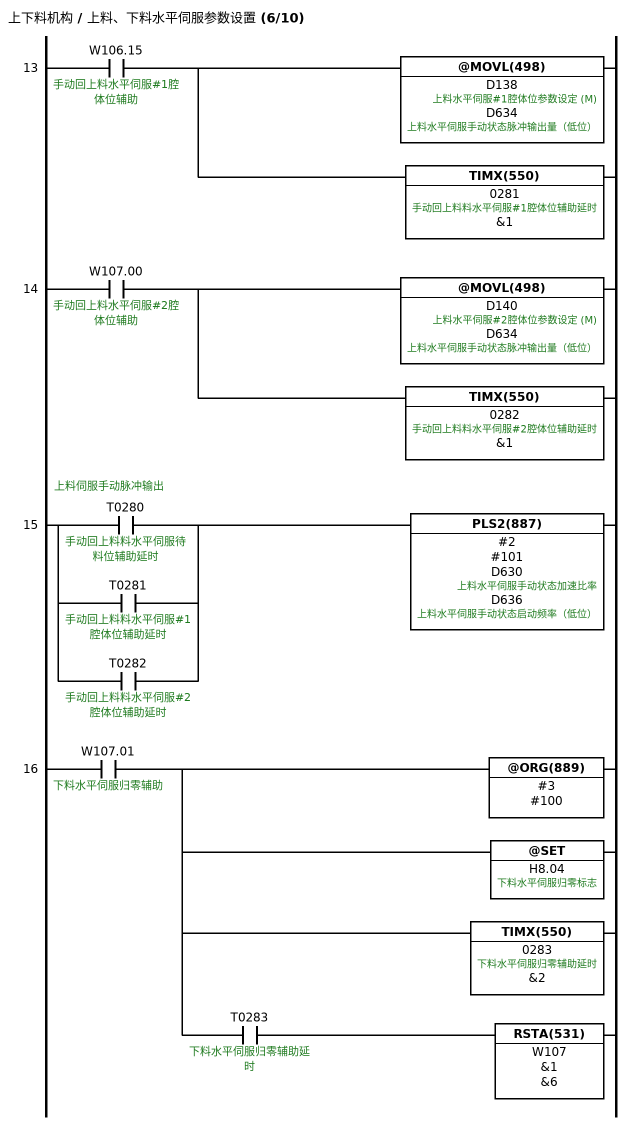
; [picture p216: 上下料机构 / 上料、下料水平伺服参数设置, rungs 13-16]
; rung 13
LD W106.15  ; 手动回上料水平伺服#1腔体位辅助
@MOVL(498) D138 D634  ; 上料水平伺服#1腔体位参数设定 (M), 上料水平伺服手动状态脉冲输出量（低位）
TIMX(550) 0281 &1  ; 手动回上料料水平伺服#1腔体位辅助延时
; rung 14
LD W107.00  ; 手动回上料水平伺服#2腔体位辅助
@MOVL(498) D140 D634  ; 上料水平伺服#2腔体位参数设定 (M), 上料水平伺服手动状态脉冲输出量（低位）
TIMX(550) 0282 &1  ; 手动回上料料水平伺服#2腔体位辅助延时
; rung 15: 上料伺服手动脉冲输出
LD T0280  ; 手动回上料料水平伺服待料位辅助延时
OR T0281  ; 手动回上料料水平伺服#1腔体位辅助延时
OR T0282  ; 手动回上料料水平伺服#2腔体位辅助延时
PLS2(887) #2 #101 D630 D636  ; 上料水平伺服手动状态加速比率, 上料水平伺服手动状态启动频率（低位）
; rung 16
LD W107.01  ; 下料水平伺服归零辅助
@ORG(889) #3 #100
@SET H8.04  ; 下料水平伺服归零标志
TIMX(550) 0283 &2  ; 下料水平伺服归零辅助延时
AND T0283  ; 下料水平伺服归零辅助延时
RSTA(531) W107 &1 &6

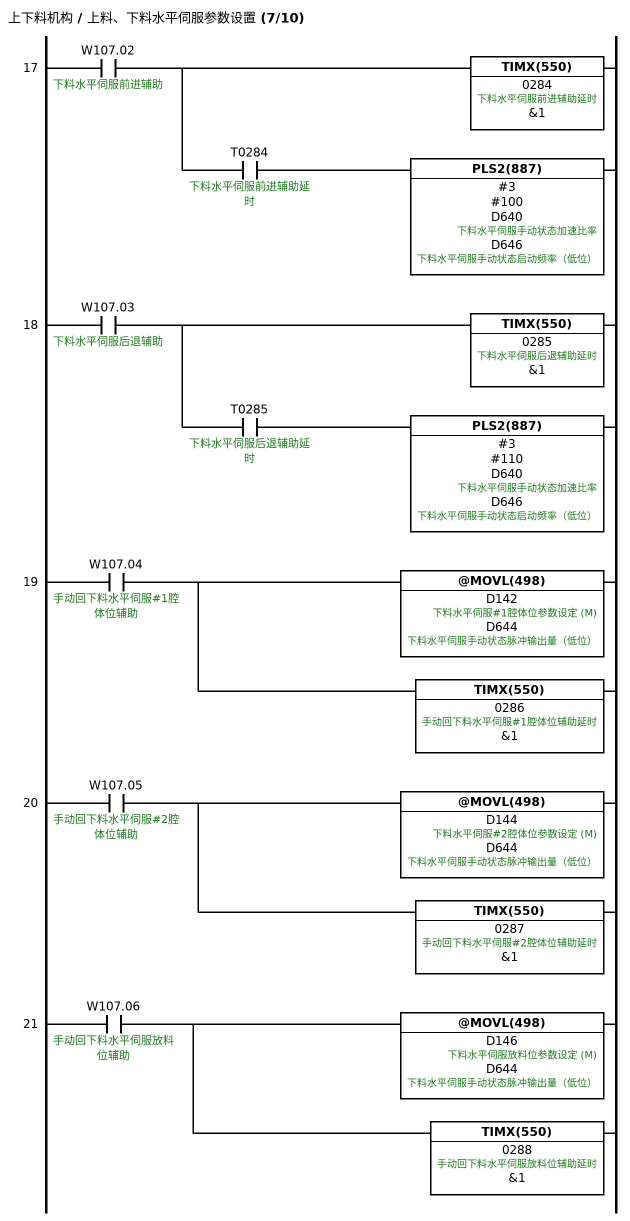
; rung 17
LD W107.02  ; 下料水平伺服前进辅助
TIMX(550) 0284 &1  ; 下料水平伺服前进辅助延时
AND T0284  ; 下料水平伺服前进辅助延时
PLS2(887) #3 #100 D640 D646  ; 下料水平伺服手动状态加速比率, 下料水平伺服手动状态启动频率（低位）
; rung 18
LD W107.03  ; 下料水平伺服后退辅助
TIMX(550) 0285 &1  ; 下料水平伺服后退辅助延时
AND T0285  ; 下料水平伺服后退辅助延时
PLS2(887) #3 #110 D640 D646  ; 下料水平伺服手动状态加速比率, 下料水平伺服手动状态启动频率（低位）
; rung 19
LD W107.04  ; 手动回下料水平伺服#1腔体位辅助
@MOVL(498) D142 D644  ; 下料水平伺服#1腔体位参数设定 (M), 下料水平伺服手动状态脉冲输出量（低位）
TIMX(550) 0286 &1  ; 手动回下料水平伺服#1腔体位辅助延时
; rung 20
LD W107.05  ; 手动回下料水平伺服#2腔体位辅助
@MOVL(498) D144 D644  ; 下料水平伺服#2腔体位参数设定 (M), 下料水平伺服手动状态脉冲输出量（低位）
TIMX(550) 0287 &1  ; 手动回下料水平伺服#2腔体位辅助延时
; rung 21
LD W107.06  ; 手动回下料水平伺服放料位辅助
@MOVL(498) D146 D644  ; 下料水平伺服放料位参数设定 (M), 下料水平伺服手动状态脉冲输出量（低位）
TIMX(550) 0288 &1  ; 手动回下料水平伺服放料位辅助延时

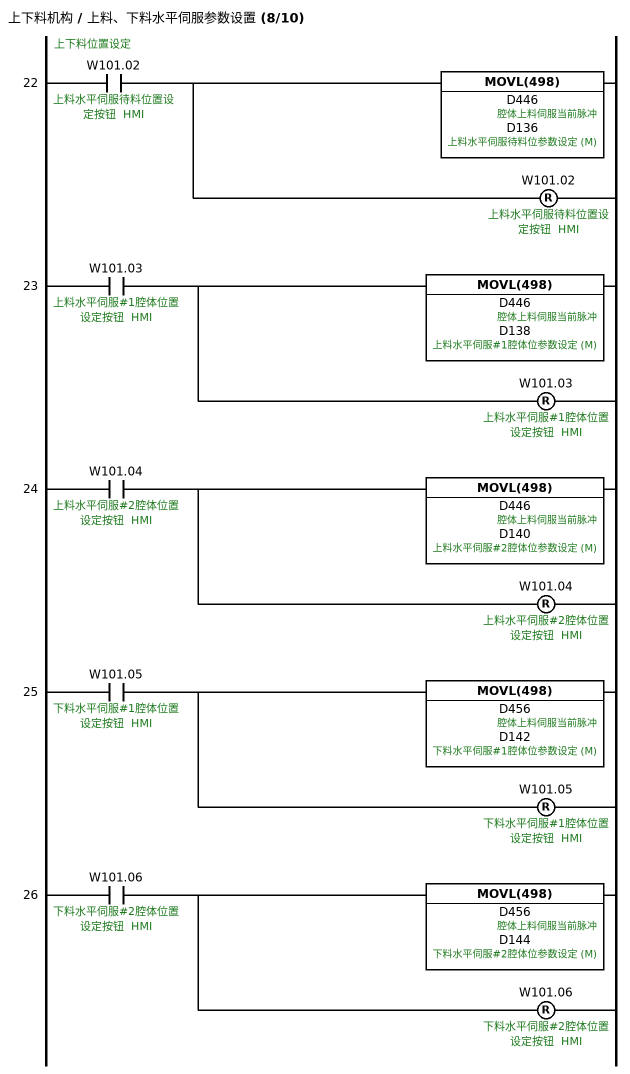
; rung 22: 上下料位置设定
LD W101.02  ; 上料水平伺服待料位置设定按钮  HMI
MOVL(498) D446 D136  ; 腔体上料伺服当前脉冲, 上料水平伺服待料位参数设定 (M)
RSET W101.02  ; 上料水平伺服待料位置设定按钮  HMI
; rung 23
LD W101.03  ; 上料水平伺服#1腔体位置设定按钮  HMI
MOVL(498) D446 D138  ; 腔体上料伺服当前脉冲, 上料水平伺服#1腔体位参数设定 (M)
RSET W101.03  ; 上料水平伺服#1腔体位置设定按钮  HMI
; rung 24
LD W101.04  ; 上料水平伺服#2腔体位置设定按钮  HMI
MOVL(498) D446 D140  ; 腔体上料伺服当前脉冲, 上料水平伺服#2腔体位参数设定 (M)
RSET W101.04  ; 上料水平伺服#2腔体位置设定按钮  HMI
; rung 25
LD W101.05  ; 下料水平伺服#1腔体位置设定按钮  HMI
MOVL(498) D456 D142  ; 腔体上料伺服当前脉冲, 下料水平伺服#1腔体位参数设定 (M)
RSET W101.05  ; 下料水平伺服#1腔体位置设定按钮  HMI
; rung 26
LD W101.06  ; 下料水平伺服#2腔体位置设定按钮  HMI
MOVL(498) D456 D144  ; 腔体上料伺服当前脉冲, 下料水平伺服#2腔体位参数设定 (M)
RSET W101.06  ; 下料水平伺服#2腔体位置设定按钮  HMI

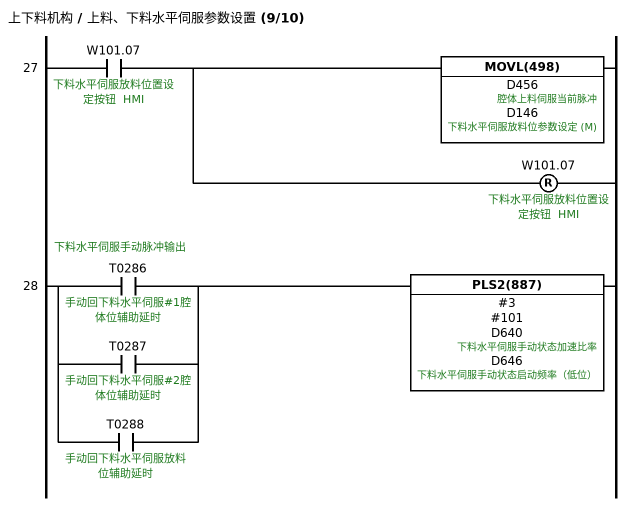
; rung 27
LD W101.07  ; 下料水平伺服放料位置设定按钮  HMI
MOVL(498) D456 D146  ; 腔体上料伺服当前脉冲, 下料水平伺服放料位参数设定 (M)
RSET W101.07  ; 下料水平伺服放料位置设定按钮  HMI
; rung 28: 下料水平伺服手动脉冲输出
LD T0286  ; 手动回下料水平伺服#1腔体位辅助延时
OR T0287  ; 手动回下料水平伺服#2腔体位辅助延时
OR T0288  ; 手动回下料水平伺服放料位辅助延时
PLS2(887) #3 #101 D640 D646  ; 下料水平伺服手动状态加速比率, 下料水平伺服手动状态启动频率（低位）

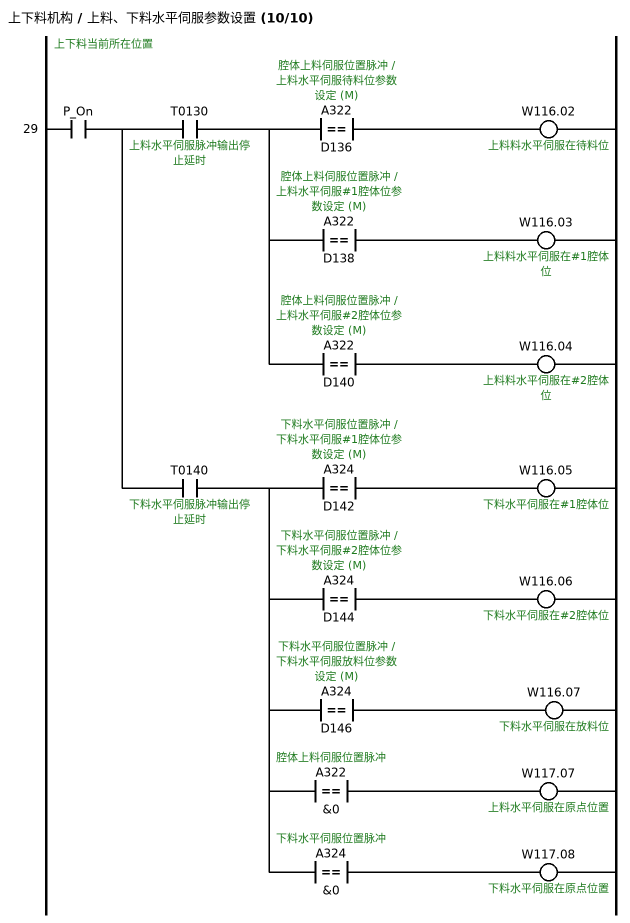
; rung 29: 上下料当前所在位置
LD P_On
OUT TR0
AND T0130  ; 上料水平伺服脉冲输出停止延时
OUT TR1
AND=SL(303) A322 D136  ; 腔体上料伺服位置脉冲, 上料水平伺服待料位参数设定 (M)
OUT W116.02  ; 上料料水平伺服在待料位
LD TR1
AND=SL(303) A322 D138  ; 腔体上料伺服位置脉冲, 上料水平伺服#1腔体位参数设定 (M)
OUT W116.03  ; 上料料水平伺服在#1腔体位
LD TR1
AND=SL(303) A322 D140  ; 腔体上料伺服位置脉冲, 上料水平伺服#2腔体位参数设定 (M)
OUT W116.04  ; 上料料水平伺服在#2腔体位
LD TR0
AND T0140  ; 下料水平伺服脉冲输出停止延时
OUT TR0
AND=SL(303) A324 D142  ; 下料水平伺服位置脉冲, 下料水平伺服#1腔体位参数设定 (M)
OUT W116.05  ; 下料水平伺服在#1腔体位
LD TR0
AND=SL(303) A324 D144  ; 下料水平伺服位置脉冲, 下料水平伺服#2腔体位参数设定 (M)
OUT W116.06  ; 下料水平伺服在#2腔体位
LD TR0
AND=SL(303) A324 D146  ; 下料水平伺服位置脉冲, 下料水平伺服放料位参数设定 (M)
OUT W116.07  ; 下料水平伺服在放料位
LD TR0
AND=SL(303) A322 &0  ; 腔体上料伺服位置脉冲
OUT W117.07  ; 上料水平伺服在原点位置
LD TR0
AND=SL(303) A324 &0  ; 下料水平伺服位置脉冲
OUT W117.08  ; 下料水平伺服在原点位置

### Section 工站复位

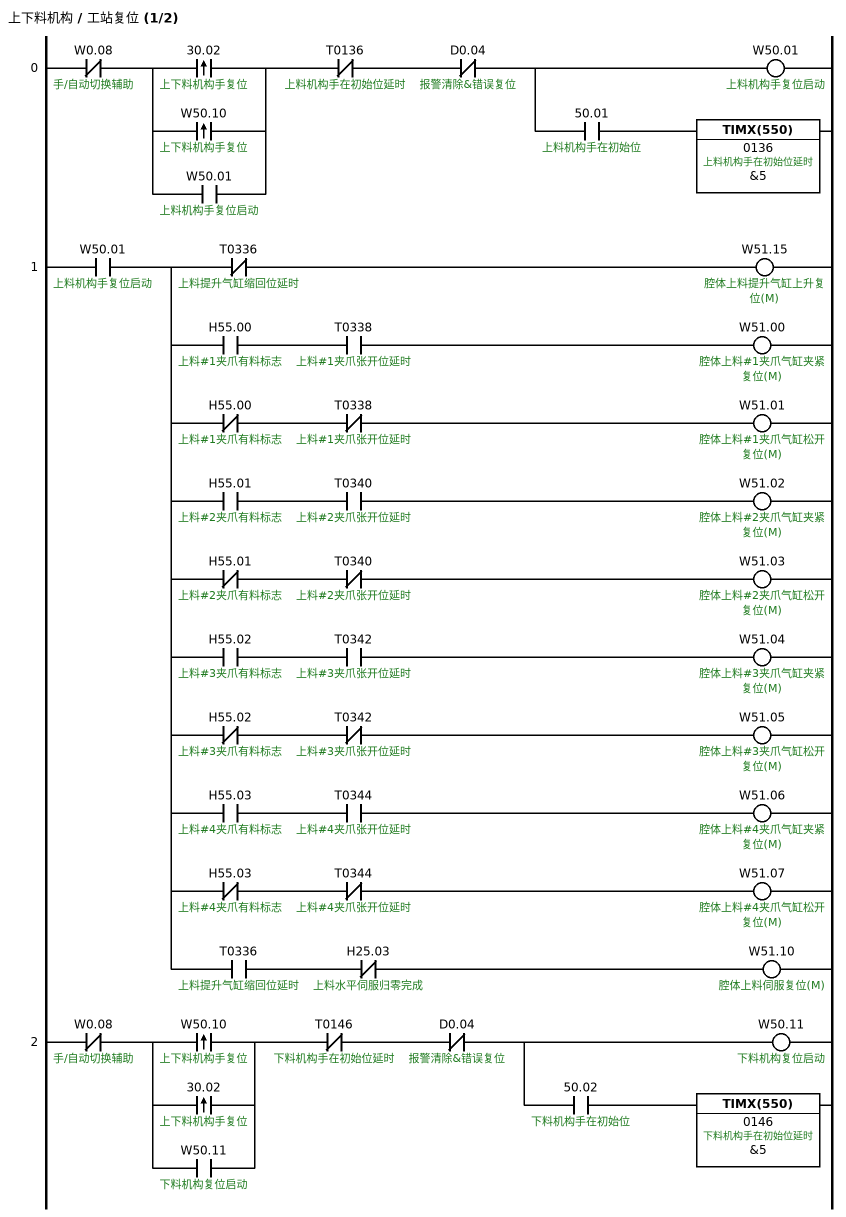
; rung 0
LDNOT W0.08  ; 手/自动切换辅助
@LD 30.02  ; 上下料机构手复位
@OR W50.10  ; 上下料机构手复位
OR W50.01  ; 上料机构手复位启动
ANDLD
ANDNOT T0136  ; 上料机构手在初始位延时
ANDNOT D0.04  ; 报警清除&错误复位
OUT W50.01  ; 上料机构手复位启动
AND 50.01  ; 上料机构手在初始位
TIMX(550) 0136 &5  ; 上料机构手在初始位延时
; rung 1
LD W50.01  ; 上料机构手复位启动
OUT TR0
ANDNOT T0336  ; 上料提升气缸缩回位延时
OUT W51.15  ; 腔体上料提升气缸上升复位(M)
LD TR0
AND H55.00  ; 上料#1夹爪有料标志
AND T0338  ; 上料#1夹爪张开位延时
OUT W51.00  ; 腔体上料#1夹爪气缸夹紧复位(M)
LD TR0
ANDNOT H55.00  ; 上料#1夹爪有料标志
ANDNOT T0338  ; 上料#1夹爪张开位延时
OUT W51.01  ; 腔体上料#1夹爪气缸松开复位(M)
LD TR0
AND H55.01  ; 上料#2夹爪有料标志
AND T0340  ; 上料#2夹爪张开位延时
OUT W51.02  ; 腔体上料#2夹爪气缸夹紧复位(M)
LD TR0
ANDNOT H55.01  ; 上料#2夹爪有料标志
ANDNOT T0340  ; 上料#2夹爪张开位延时
OUT W51.03  ; 腔体上料#2夹爪气缸松开复位(M)
LD TR0
AND H55.02  ; 上料#3夹爪有料标志
AND T0342  ; 上料#3夹爪张开位延时
OUT W51.04  ; 腔体上料#3夹爪气缸夹紧复位(M)
LD TR0
ANDNOT H55.02  ; 上料#3夹爪有料标志
ANDNOT T0342  ; 上料#3夹爪张开位延时
OUT W51.05  ; 腔体上料#3夹爪气缸松开复位(M)
LD TR0
AND H55.03  ; 上料#4夹爪有料标志
AND T0344  ; 上料#4夹爪张开位延时
OUT W51.06  ; 腔体上料#4夹爪气缸夹紧复位(M)
LD TR0
ANDNOT H55.03  ; 上料#4夹爪有料标志
ANDNOT T0344  ; 上料#4夹爪张开位延时
OUT W51.07  ; 腔体上料#4夹爪气缸松开复位(M)
LD TR0
AND T0336  ; 上料提升气缸缩回位延时
ANDNOT H25.03  ; 上料水平伺服归零完成
OUT W51.10  ; 腔体上料伺服复位(M)
; rung 2
LDNOT W0.08  ; 手/自动切换辅助
@LD W50.10  ; 上下料机构手复位
@OR 30.02  ; 上下料机构手复位
OR W50.11  ; 下料机构复位启动
ANDLD
ANDNOT T0146  ; 下料机构手在初始位延时
ANDNOT D0.04  ; 报警清除&错误复位
OUT W50.11  ; 下料机构复位启动
AND 50.02  ; 下料机构手在初始位
TIMX(550) 0146 &5  ; 下料机构手在初始位延时

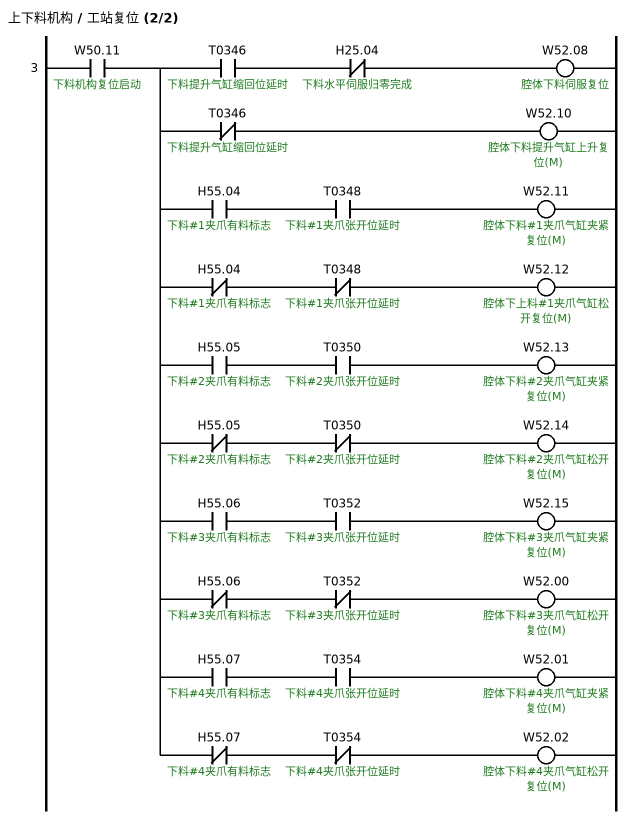
; rung 3
LD W50.11  ; 下料机构复位启动
OUT TR0
AND T0346  ; 下料提升气缸缩回位延时
ANDNOT H25.04  ; 下料水平伺服归零完成
OUT W52.08  ; 腔体下料伺服复位
LD TR0
ANDNOT T0346  ; 下料提升气缸缩回位延时
OUT W52.10  ; 腔体下料提升气缸上升复位(M)
LD TR0
AND H55.04  ; 下料#1夹爪有料标志
AND T0348  ; 下料#1夹爪张开位延时
OUT W52.11  ; 腔体下料#1夹爪气缸夹紧复位(M)
LD TR0
ANDNOT H55.04  ; 下料#1夹爪有料标志
ANDNOT T0348  ; 下料#1夹爪张开位延时
OUT W52.12  ; 腔体下上料#1夹爪气缸松开复位(M)
LD TR0
AND H55.05  ; 下料#2夹爪有料标志
AND T0350  ; 下料#2夹爪张开位延时
OUT W52.13  ; 腔体下料#2夹爪气缸夹紧复位(M)
LD TR0
ANDNOT H55.05  ; 下料#2夹爪有料标志
ANDNOT T0350  ; 下料#2夹爪张开位延时
OUT W52.14  ; 腔体下料#2夹爪气缸松开复位(M)
LD TR0
AND H55.06  ; 下料#3夹爪有料标志
AND T0352  ; 下料#3夹爪张开位延时
OUT W52.15  ; 腔体下料#3夹爪气缸夹紧复位(M)
LD TR0
ANDNOT H55.06  ; 下料#3夹爪有料标志
ANDNOT T0352  ; 下料#3夹爪张开位延时
OUT W52.00  ; 腔体下料#3夹爪气缸松开复位(M)
LD TR0
AND H55.07  ; 下料#4夹爪有料标志
AND T0354  ; 下料#4夹爪张开位延时
OUT W52.01  ; 腔体下料#4夹爪气缸夹紧复位(M)
LD TR0
ANDNOT H55.07  ; 下料#4夹爪有料标志
ANDNOT T0354  ; 下料#4夹爪张开位延时
OUT W52.02  ; 腔体下料#4夹爪气缸松开复位(M)

### Section 指示灯

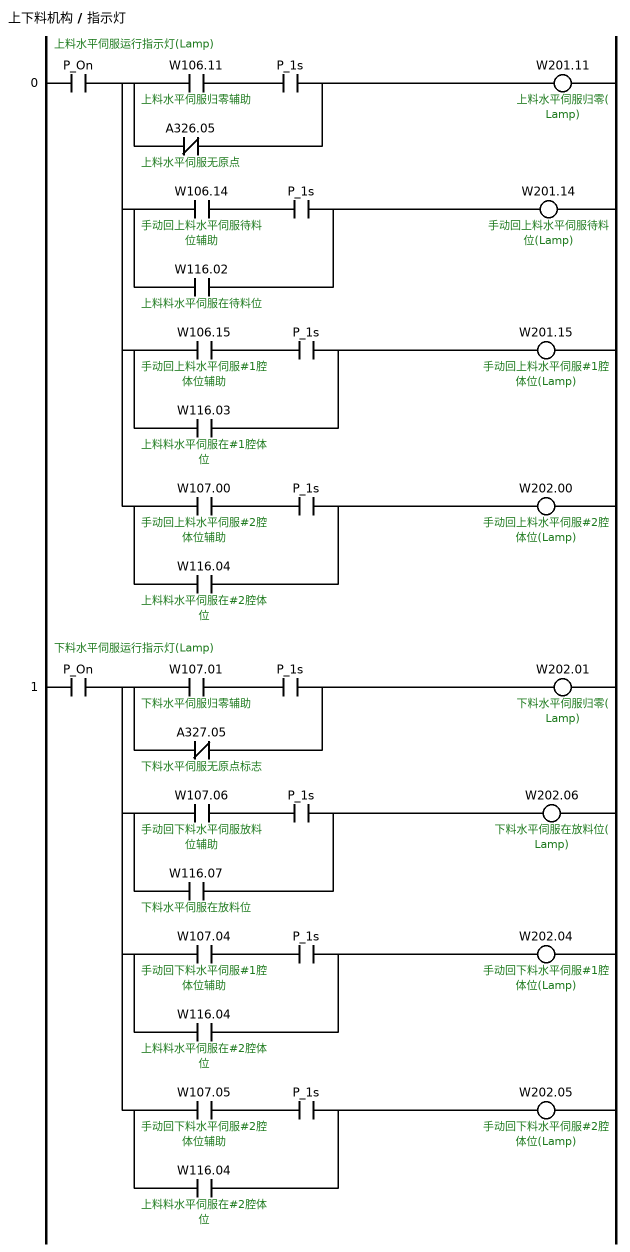
; rung 0: 上料水平伺服运行指示灯(Lamp)
LD P_On
OUT TR0
LD W106.11  ; 上料水平伺服归零辅助
AND P_1s
ORNOT A326.05  ; 上料水平伺服无原点
ANDLD
OUT W201.11  ; 上料水平伺服归零(Lamp)
LD TR0
LD W106.14  ; 手动回上料水平伺服待料位辅助
AND P_1s
OR W116.02  ; 上料料水平伺服在待料位
ANDLD
OUT W201.14  ; 手动回上料水平伺服待料位(Lamp)
LD TR0
LD W106.15  ; 手动回上料水平伺服#1腔体位辅助
AND P_1s
OR W116.03  ; 上料料水平伺服在#1腔体位
ANDLD
OUT W201.15  ; 手动回上料水平伺服#1腔体位(Lamp)
LD TR0
LD W107.00  ; 手动回上料水平伺服#2腔体位辅助
AND P_1s
OR W116.04  ; 上料料水平伺服在#2腔体位
ANDLD
OUT W202.00  ; 手动回上料水平伺服#2腔体位(Lamp)
; rung 1: 下料水平伺服运行指示灯(Lamp)
LD P_On
OUT TR0
LD W107.01  ; 下料水平伺服归零辅助
AND P_1s
ORNOT A327.05  ; 下料水平伺服无原点标志
ANDLD
OUT W202.01  ; 下料水平伺服归零(Lamp)
LD TR0
LD W107.06  ; 手动回下料水平伺服放料位辅助
AND P_1s
OR W116.07  ; 下料水平伺服在放料位
ANDLD
OUT W202.06  ; 下料水平伺服在放料位(Lamp)
LD TR0
LD W107.04  ; 手动回下料水平伺服#1腔体位辅助
AND P_1s
OR W116.04  ; 上料料水平伺服在#2腔体位
ANDLD
OUT W202.04  ; 手动回下料水平伺服#1腔体位(Lamp)
LD TR0
LD W107.05  ; 手动回下料水平伺服#2腔体位辅助
AND P_1s
OR W116.04  ; 上料料水平伺服在#2腔体位
ANDLD
OUT W202.05  ; 手动回下料水平伺服#2腔体位(Lamp)

### Section 临时

### Section END
; rung 0
END(001)

## Program 腔体机构 (cyclic task 3)

### Section 真空值及漏率转换

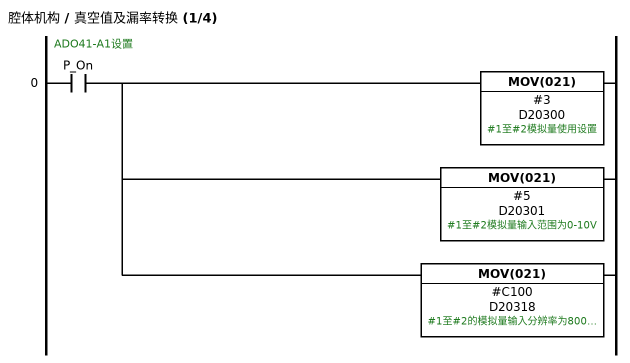
; rung 0: ADO41-A1设置
LD P_On
MOV(021) #3 D20300  ; #1至#2模拟量使用设置
MOV(021) #5 D20301  ; #1至#2模拟量输入范围为0-10V
MOV(021) #C100 D20318  ; #1至#2的模拟量输入分辨率为8000   普通模式

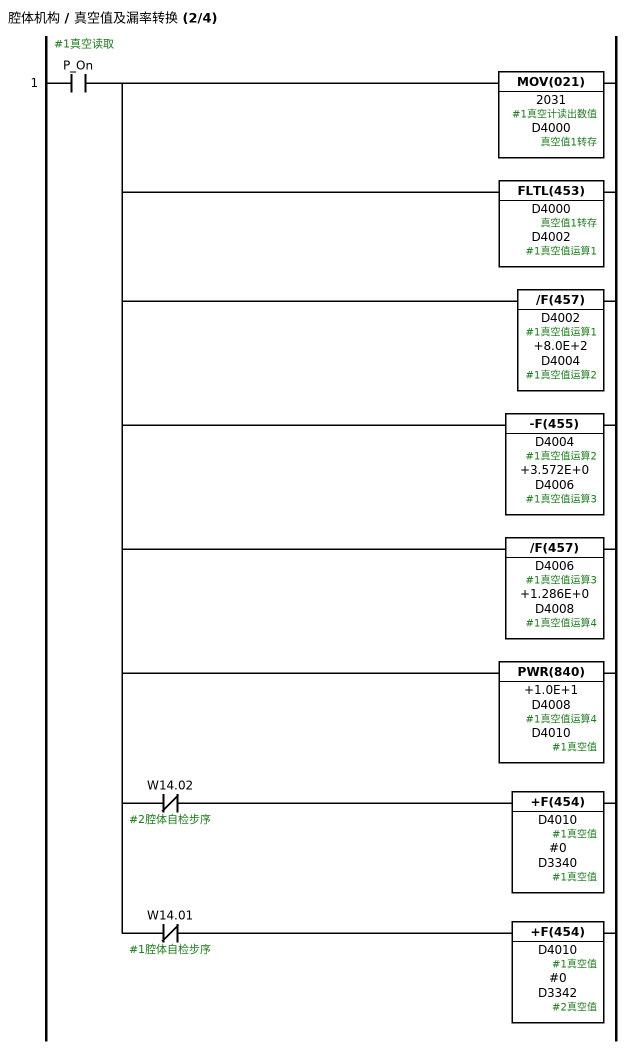
; rung 1: #1真空读取
LD P_On
OUT TR0
MOV(021) 2031 D4000  ; #1真空计读出数值, 真空值1转存
FLTL(453) D4000 D4002  ; 真空值1转存, #1真空值运算1
/F(457) D4002 +8.0E+2 D4004  ; #1真空值运算1, #1真空值运算2
-F(455) D4004 +3.572E+0 D4006  ; #1真空值运算2, #1真空值运算3
/F(457) D4006 +1.286E+0 D4008  ; #1真空值运算3, #1真空值运算4
PWR(840) +1.0E+1 D4008 D4010  ; #1真空值运算4, #1真空值
ANDNOT W14.02  ; #2腔体自检步序
+F(454) D4010 #0 D3340  ; #1真空值
LD TR0
ANDNOT W14.01  ; #1腔体自检步序
+F(454) D4010 #0 D3342  ; #1真空值, #2真空值

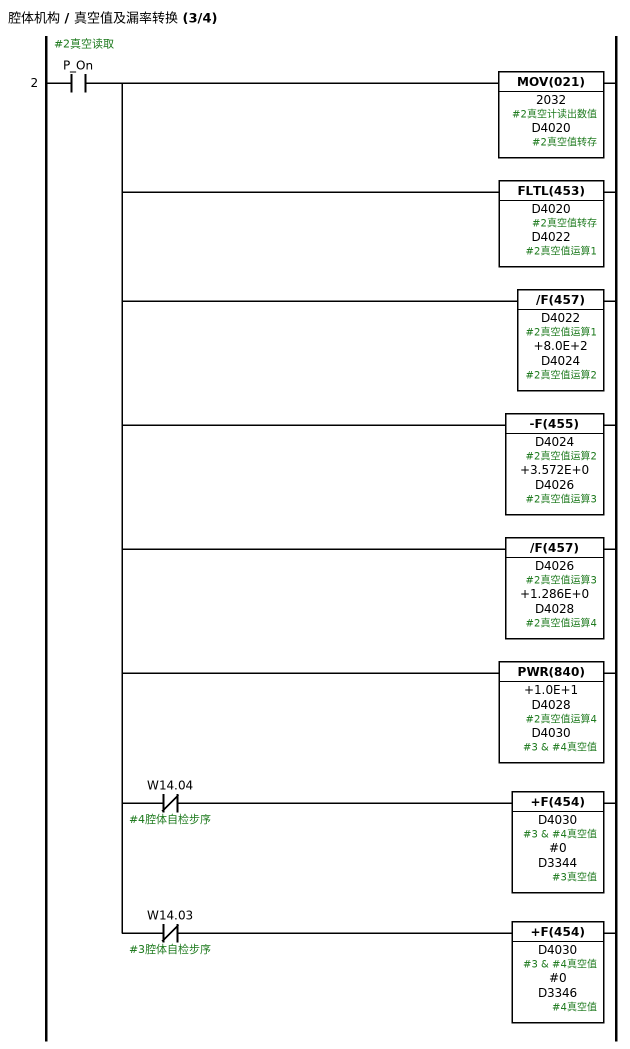
; rung 2: #2真空读取
LD P_On
OUT TR0
MOV(021) 2032 D4020  ; #2真空计读出数值, #2真空值转存
FLTL(453) D4020 D4022  ; #2真空值转存, #2真空值运算1
/F(457) D4022 +8.0E+2 D4024  ; #2真空值运算1, #2真空值运算2
-F(455) D4024 +3.572E+0 D4026  ; #2真空值运算2, #2真空值运算3
/F(457) D4026 +1.286E+0 D4028  ; #2真空值运算3, #2真空值运算4
PWR(840) +1.0E+1 D4028 D4030  ; #2真空值运算4, #3 & #4真空值
ANDNOT W14.04  ; #4腔体自检步序
+F(454) D4030 #0 D3344  ; #3 & #4真空值, #3真空值
LD TR0
ANDNOT W14.03  ; #3腔体自检步序
+F(454) D4030 #0 D3346  ; #3 & #4真空值, #4真空值

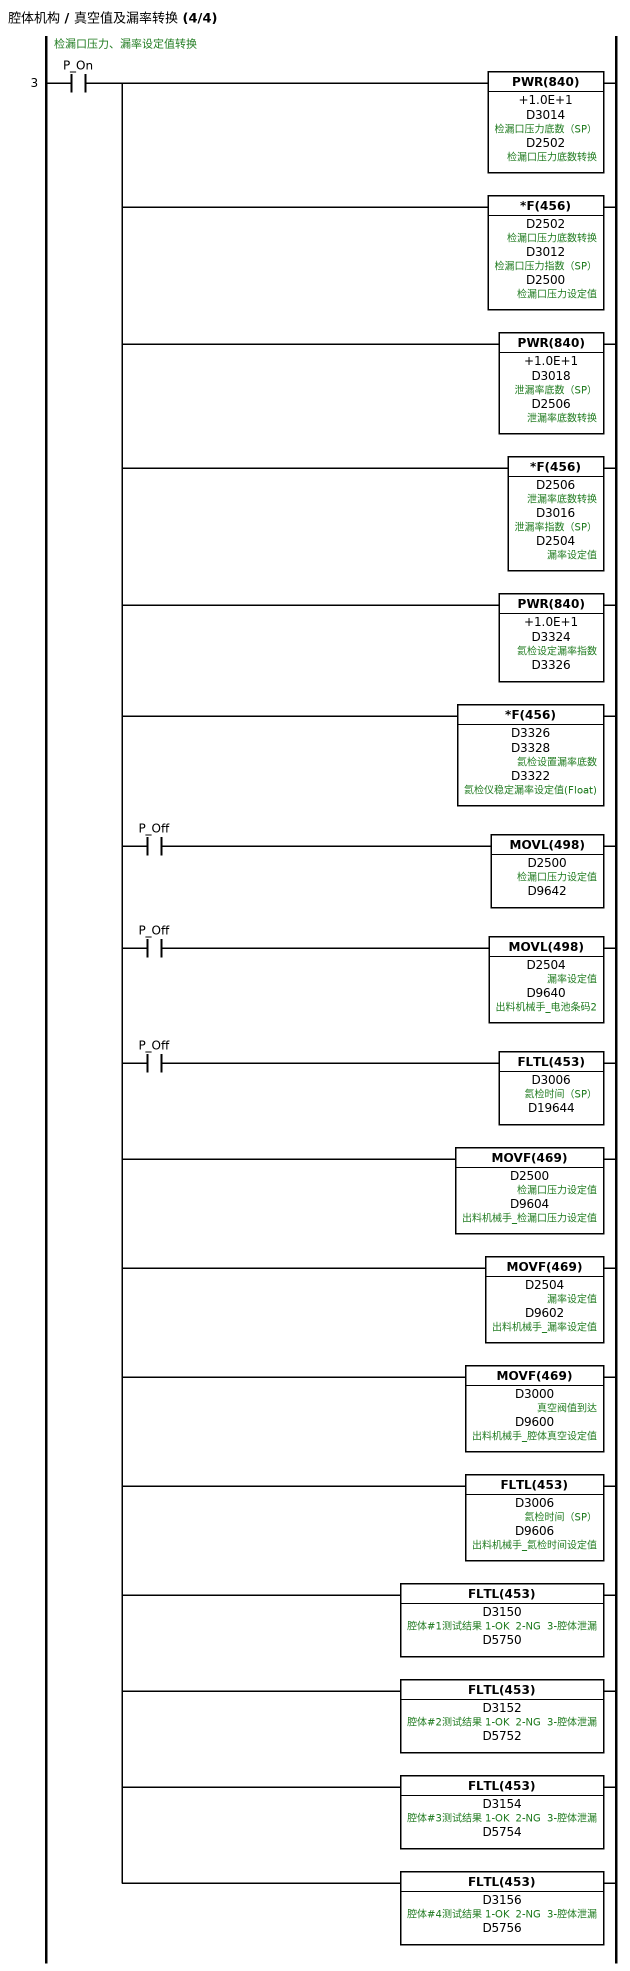
; rung 3: 检漏口压力、漏率设定值转换
LD P_On
OUT TR0
PWR(840) +1.0E+1 D3014 D2502  ; 检漏口压力底数（SP）, 检漏口压力底数转换
*F(456) D2502 D3012 D2500  ; 检漏口压力底数转换, 检漏口压力指数（SP）, 检漏口压力设定值
PWR(840) +1.0E+1 D3018 D2506  ; 泄漏率底数（SP）, 泄漏率底数转换
*F(456) D2506 D3016 D2504  ; 泄漏率底数转换, 泄漏率指数（SP）, 漏率设定值
PWR(840) +1.0E+1 D3324 D3326  ; 氦检设定漏率指数
*F(456) D3326 D3328 D3322  ; 氦检设置漏率底数, 氦检仪稳定漏率设定值(Float)
AND P_Off
MOVL(498) D2500 D9642  ; 检漏口压力设定值
LD TR0
AND P_Off
MOVL(498) D2504 D9640  ; 漏率设定值, 出料机械手_电池条码2
LD TR0
AND P_Off
FLTL(453) D3006 D19644  ; 氦检时间（SP）
LD TR0
MOVF(469) D2500 D9604  ; 检漏口压力设定值, 出料机械手_检漏口压力设定值
MOVF(469) D2504 D9602  ; 漏率设定值, 出料机械手_漏率设定值
MOVF(469) D3000 D9600  ; 真空阀值到达, 出料机械手_腔体真空设定值
FLTL(453) D3006 D9606  ; 氦检时间（SP）, 出料机械手_氦检时间设定值
FLTL(453) D3150 D5750  ; 腔体#1测试结果 1-OK  2-NG  3-腔体泄漏
FLTL(453) D3152 D5752  ; 腔体#2测试结果 1-OK  2-NG  3-腔体泄漏
FLTL(453) D3154 D5754  ; 腔体#3测试结果 1-OK  2-NG  3-腔体泄漏
FLTL(453) D3156 D5756  ; 腔体#4测试结果 1-OK  2-NG  3-腔体泄漏

### Section 氦检

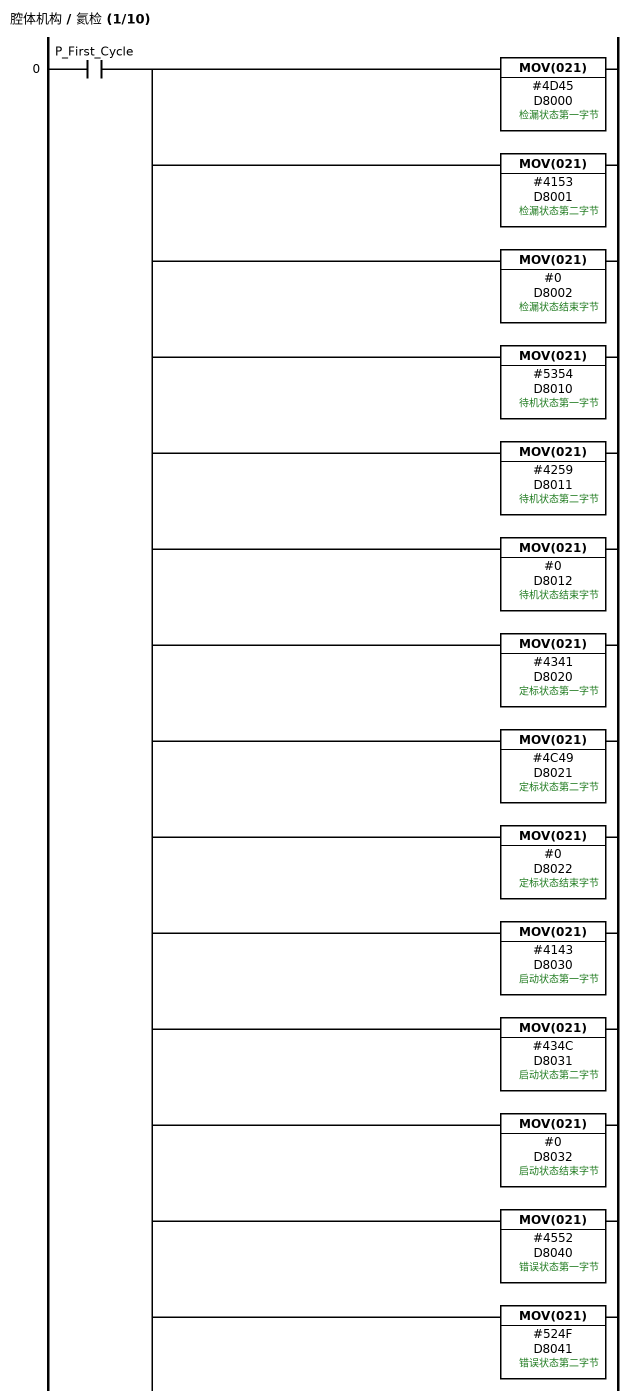

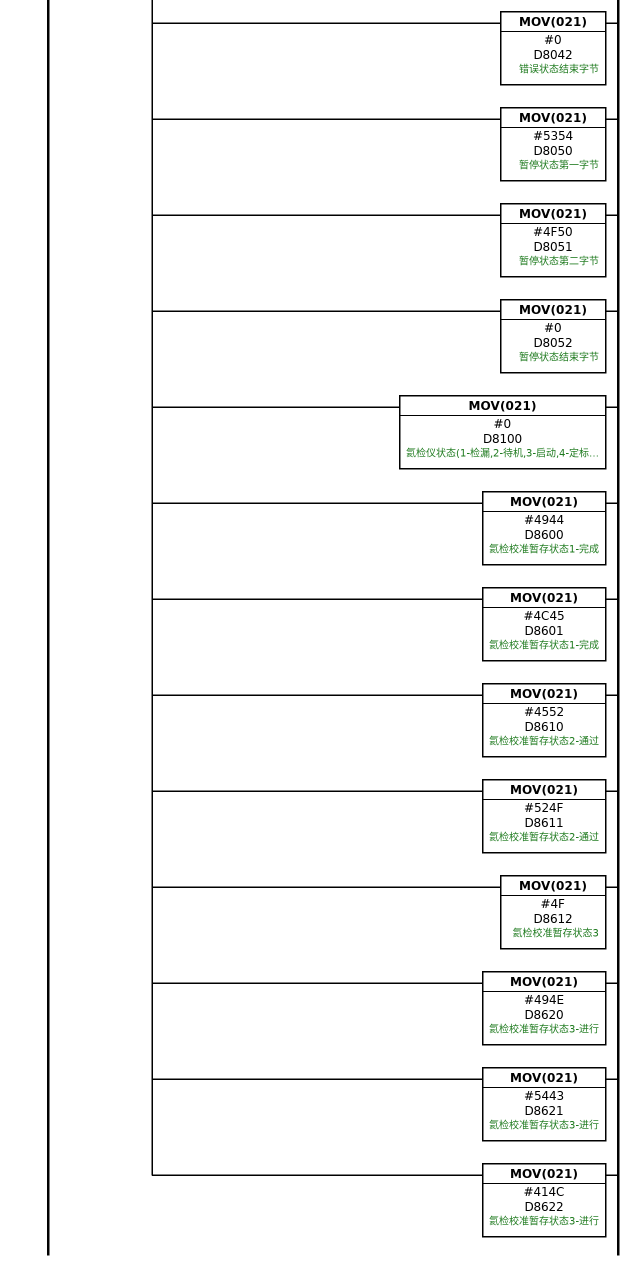
; rung 0
LD P_First_Cycle
MOV(021) #4D45 D8000  ; 检漏状态第一字节
MOV(021) #4153 D8001  ; 检漏状态第二字节
MOV(021) #0 D8002  ; 检漏状态结束字节
MOV(021) #5354 D8010  ; 待机状态第一字节
MOV(021) #4259 D8011  ; 待机状态第二字节
MOV(021) #0 D8012  ; 待机状态结束字节
MOV(021) #4341 D8020  ; 定标状态第一字节
MOV(021) #4C49 D8021  ; 定标状态第二字节
MOV(021) #0 D8022  ; 定标状态结束字节
MOV(021) #4143 D8030  ; 启动状态第一字节
MOV(021) #434C D8031  ; 启动状态第二字节
MOV(021) #0 D8032  ; 启动状态结束字节
MOV(021) #4552 D8040  ; 错误状态第一字节
MOV(021) #524F D8041  ; 错误状态第二字节
MOV(021) #0 D8042  ; 错误状态结束字节
MOV(021) #5354 D8050  ; 暂停状态第一字节
MOV(021) #4F50 D8051  ; 暂停状态第二字节
MOV(021) #0 D8052  ; 暂停状态结束字节
MOV(021) #0 D8100  ; 氦检仪状态(1-检漏,2-待机,3-启动,4-定标,5-错误,6-暂停)
MOV(021) #4944 D8600  ; 氦检校准暂存状态1-完成
MOV(021) #4C45 D8601  ; 氦检校准暂存状态1-完成
MOV(021) #4552 D8610  ; 氦检校准暂存状态2-通过
MOV(021) #524F D8611  ; 氦检校准暂存状态2-通过
MOV(021) #4F D8612  ; 氦检校准暂存状态3
MOV(021) #494E D8620  ; 氦检校准暂存状态3-进行
MOV(021) #5443 D8621  ; 氦检校准暂存状态3-进行
MOV(021) #414C D8622  ; 氦检校准暂存状态3-进行

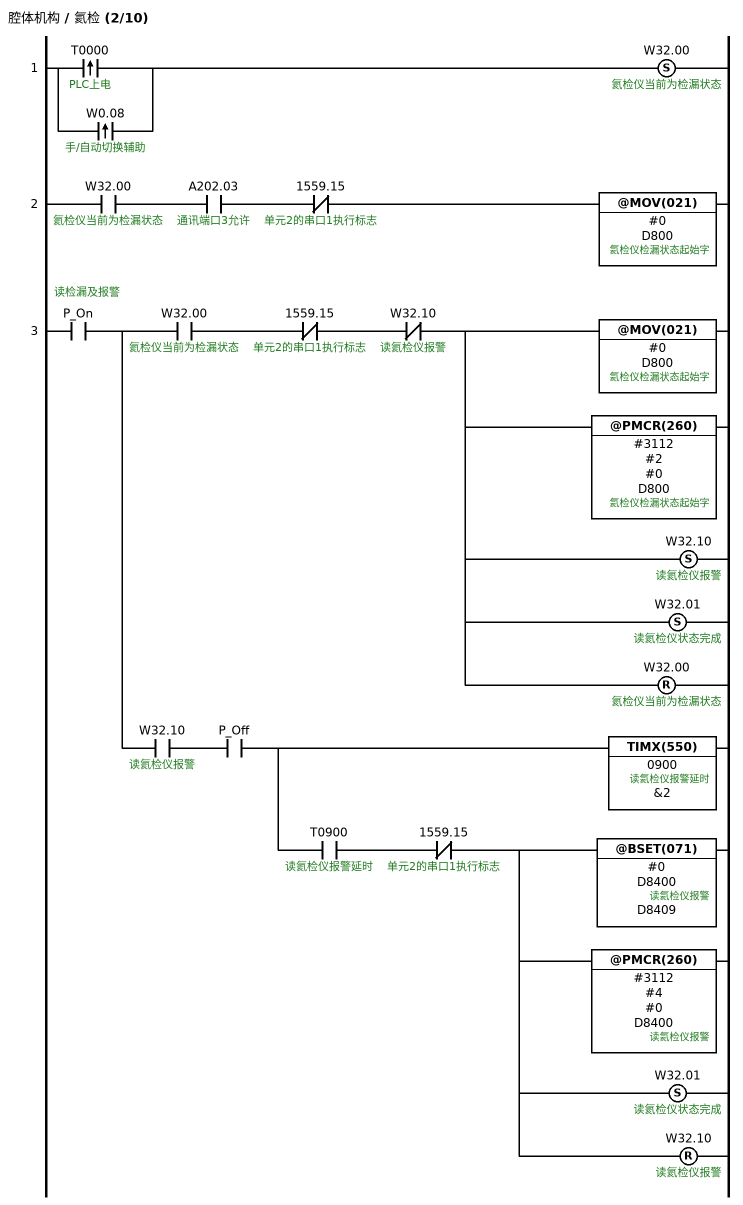
; rung 1
@LD T0000  ; PLC上电
@OR W0.08  ; 手/自动切换辅助
SET W32.00  ; 氦检仪当前为检漏状态
; rung 2
LD W32.00  ; 氦检仪当前为检漏状态
AND A202.03  ; 通讯端口3允许
ANDNOT 1559.15  ; 单元2的串口1执行标志
@MOV(021) #0 D800  ; 氦检仪检漏状态起始字
; rung 3: 读检漏及报警
LD P_On
OUT TR0
AND W32.00  ; 氦检仪当前为检漏状态
ANDNOT 1559.15  ; 单元2的串口1执行标志
ANDNOT W32.10  ; 读氦检仪报警
@MOV(021) #0 D800  ; 氦检仪检漏状态起始字
@PMCR(260) #3112 #2 #0 D800  ; 氦检仪检漏状态起始字
SET W32.10  ; 读氦检仪报警
SET W32.01  ; 读氦检仪状态完成
RSET W32.00  ; 氦检仪当前为检漏状态
LD TR0
AND W32.10  ; 读氦检仪报警
AND P_Off
TIMX(550) 0900 &2  ; 读氦检仪报警延时
AND T0900  ; 读氦检仪报警延时
ANDNOT 1559.15  ; 单元2的串口1执行标志
@BSET(071) #0 D8400 D8409  ; 读氦检仪报警
@PMCR(260) #3112 #4 #0 D8400  ; 读氦检仪报警
SET W32.01  ; 读氦检仪状态完成
RSET W32.10  ; 读氦检仪报警

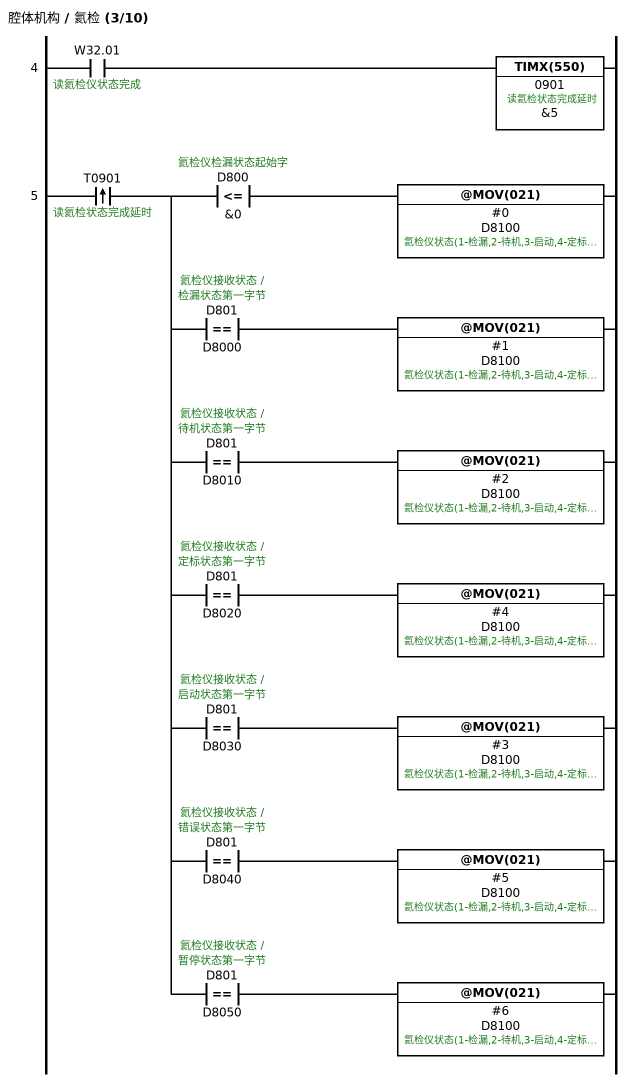
; rung 4
LD W32.01  ; 读氦检仪状态完成
TIMX(550) 0901 &5  ; 读氦检状态完成延时
; rung 5
@LD T0901  ; 读氦检状态完成延时
OUT TR0
AND<=(315) D800 &0  ; 氦检仪检漏状态起始字
@MOV(021) #0 D8100  ; 氦检仪状态(1-检漏,2-待机,3-启动,4-定标,5-错误,6-暂停)
LD TR0
AND=L(301) D801 D8000  ; 氦检仪接收状态, 检漏状态第一字节
@MOV(021) #1 D8100  ; 氦检仪状态(1-检漏,2-待机,3-启动,4-定标,5-错误,6-暂停)
LD TR0
AND=L(301) D801 D8010  ; 氦检仪接收状态, 待机状态第一字节
@MOV(021) #2 D8100  ; 氦检仪状态(1-检漏,2-待机,3-启动,4-定标,5-错误,6-暂停)
LD TR0
AND=L(301) D801 D8020  ; 氦检仪接收状态, 定标状态第一字节
@MOV(021) #4 D8100  ; 氦检仪状态(1-检漏,2-待机,3-启动,4-定标,5-错误,6-暂停)
LD TR0
AND=L(301) D801 D8030  ; 氦检仪接收状态, 启动状态第一字节
@MOV(021) #3 D8100  ; 氦检仪状态(1-检漏,2-待机,3-启动,4-定标,5-错误,6-暂停)
LD TR0
AND=L(301) D801 D8040  ; 氦检仪接收状态, 错误状态第一字节
@MOV(021) #5 D8100  ; 氦检仪状态(1-检漏,2-待机,3-启动,4-定标,5-错误,6-暂停)
LD TR0
AND=L(301) D801 D8050  ; 氦检仪接收状态, 暂停状态第一字节
@MOV(021) #6 D8100  ; 氦检仪状态(1-检漏,2-待机,3-启动,4-定标,5-错误,6-暂停)

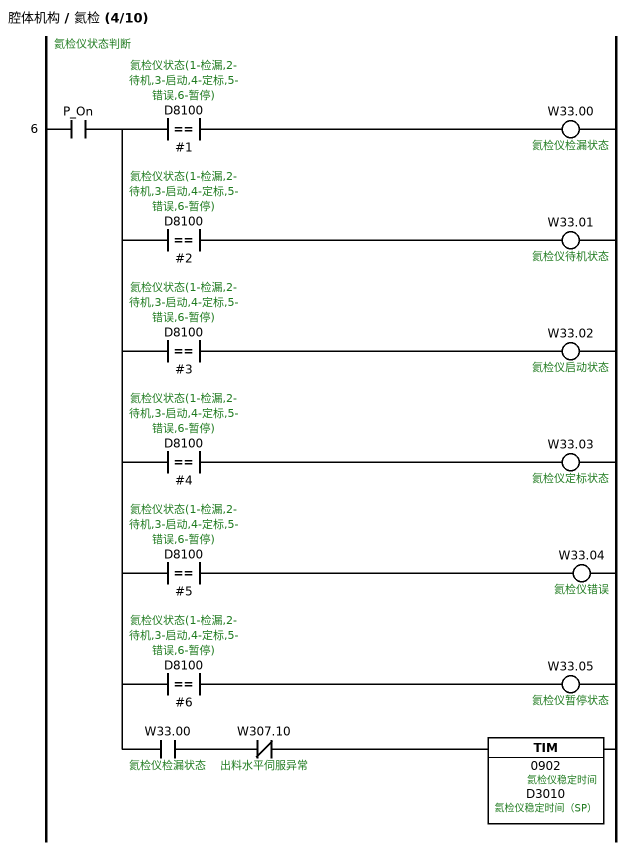
; rung 6: 氦检仪状态判断
LD P_On
OUT TR0
AND=(300) D8100 #1  ; 氦检仪状态(1-检漏,2-待机,3-启动,4-定标,5-错误,6-暂停)
OUT W33.00  ; 氦检仪检漏状态
LD TR0
AND=(300) D8100 #2  ; 氦检仪状态(1-检漏,2-待机,3-启动,4-定标,5-错误,6-暂停)
OUT W33.01  ; 氦检仪待机状态
LD TR0
AND=(300) D8100 #3  ; 氦检仪状态(1-检漏,2-待机,3-启动,4-定标,5-错误,6-暂停)
OUT W33.02  ; 氦检仪启动状态
LD TR0
AND=(300) D8100 #4  ; 氦检仪状态(1-检漏,2-待机,3-启动,4-定标,5-错误,6-暂停)
OUT W33.03  ; 氦检仪定标状态
LD TR0
AND=(300) D8100 #5  ; 氦检仪状态(1-检漏,2-待机,3-启动,4-定标,5-错误,6-暂停)
OUT W33.04  ; 氦检仪错误
LD TR0
AND=(300) D8100 #6  ; 氦检仪状态(1-检漏,2-待机,3-启动,4-定标,5-错误,6-暂停)
OUT W33.05  ; 氦检仪暂停状态
LD TR0
AND W33.00  ; 氦检仪检漏状态
ANDNOT W307.10  ; 出料水平伺服异常
TIM 0902 D3010  ; 氦检仪稳定时间（SP）, 氦检仪稳定时间

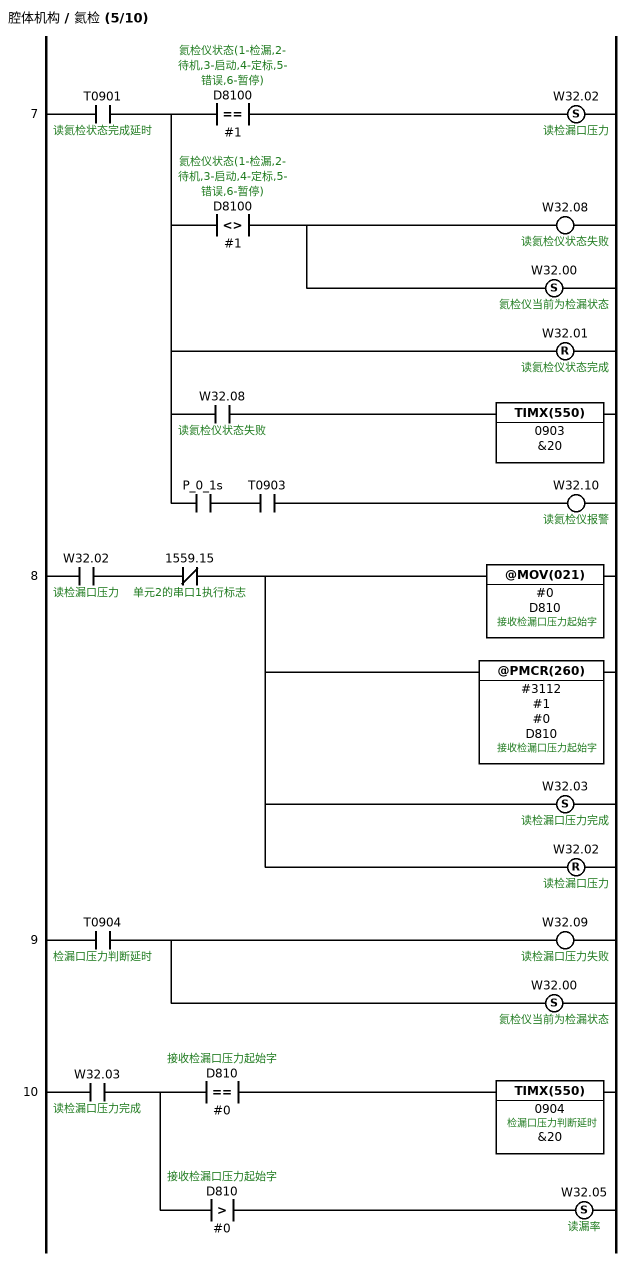
; rung 7
LD T0901  ; 读氦检状态完成延时
OUT TR0
AND=(300) D8100 #1  ; 氦检仪状态(1-检漏,2-待机,3-启动,4-定标,5-错误,6-暂停)
SET W32.02  ; 读检漏口压力
LD TR0
AND<>(305) D8100 #1  ; 氦检仪状态(1-检漏,2-待机,3-启动,4-定标,5-错误,6-暂停)
OUT W32.08  ; 读氦检仪状态失败
SET W32.00  ; 氦检仪当前为检漏状态
LD TR0
RSET W32.01  ; 读氦检仪状态完成
AND W32.08  ; 读氦检仪状态失败
TIMX(550) 0903 &20
LD TR0
AND P_0_1s
AND T0903
OUT W32.10  ; 读氦检仪报警
; rung 8
LD W32.02  ; 读检漏口压力
ANDNOT 1559.15  ; 单元2的串口1执行标志
@MOV(021) #0 D810  ; 接收检漏口压力起始字
@PMCR(260) #3112 #1 #0 D810  ; 接收检漏口压力起始字
SET W32.03  ; 读检漏口压力完成
RSET W32.02  ; 读检漏口压力
; rung 9
LD T0904  ; 检漏口压力判断延时
OUT W32.09  ; 读检漏口压力失败
SET W32.00  ; 氦检仪当前为检漏状态
; rung 10
LD W32.03  ; 读检漏口压力完成
OUT TR0
AND=(300) D810 #0  ; 接收检漏口压力起始字
TIMX(550) 0904 &20  ; 检漏口压力判断延时
LD TR0
AND>(320) D810 #0  ; 接收检漏口压力起始字
SET W32.05  ; 读漏率

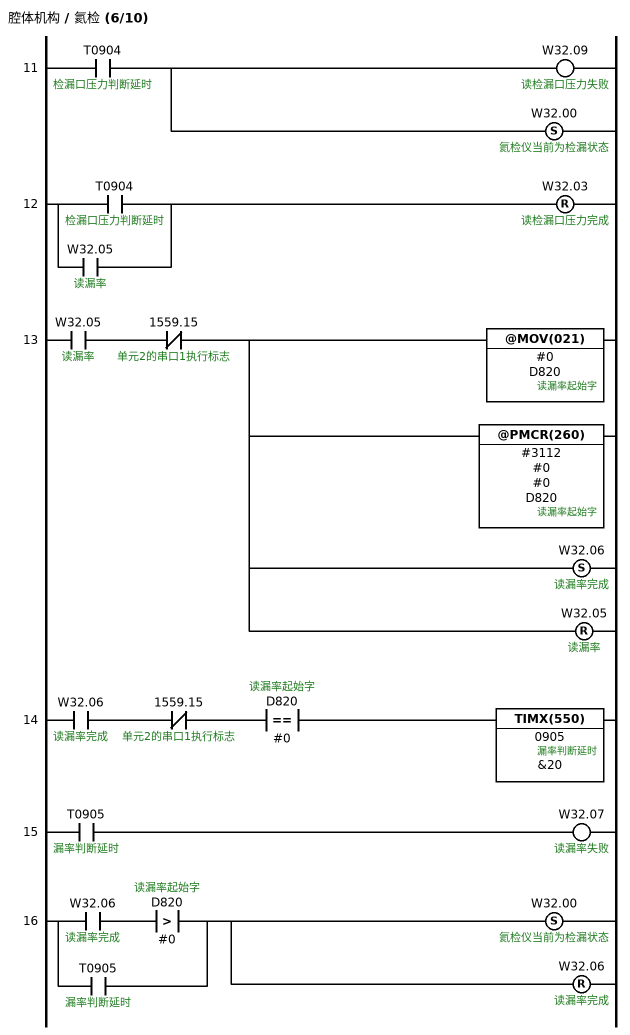
; rung 11
LD T0904  ; 检漏口压力判断延时
OUT W32.09  ; 读检漏口压力失败
SET W32.00  ; 氦检仪当前为检漏状态
; rung 12
LD T0904  ; 检漏口压力判断延时
OR W32.05  ; 读漏率
RSET W32.03  ; 读检漏口压力完成
; rung 13
LD W32.05  ; 读漏率
ANDNOT 1559.15  ; 单元2的串口1执行标志
@MOV(021) #0 D820  ; 读漏率起始字
@PMCR(260) #3112 #0 #0 D820  ; 读漏率起始字
SET W32.06  ; 读漏率完成
RSET W32.05  ; 读漏率
; rung 14
LD W32.06  ; 读漏率完成
ANDNOT 1559.15  ; 单元2的串口1执行标志
AND=(300) D820 #0  ; 读漏率起始字
TIMX(550) 0905 &20  ; 漏率判断延时
; rung 15
LD T0905  ; 漏率判断延时
OUT W32.07  ; 读漏率失败
; rung 16
LD W32.06  ; 读漏率完成
AND>(320) D820 #0  ; 读漏率起始字
OR T0905  ; 漏率判断延时
SET W32.00  ; 氦检仪当前为检漏状态
RSET W32.06  ; 读漏率完成

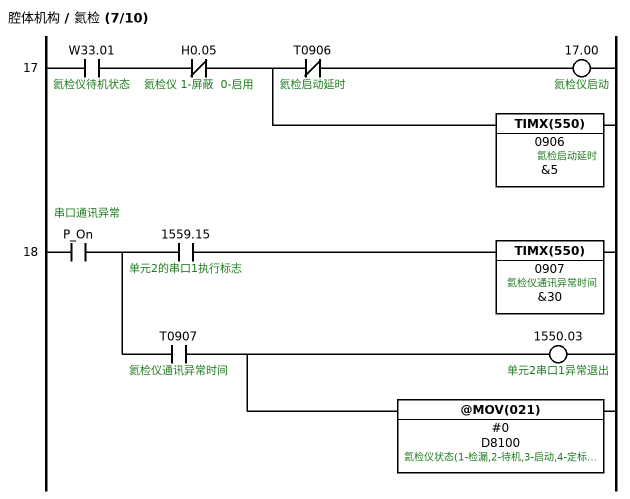
; rung 17
LD W33.01  ; 氦检仪待机状态
ANDNOT H0.05  ; 氦检仪 1-屏蔽  0-启用
OUT TR0
ANDNOT T0906  ; 氦检启动延时
OUT 17.00  ; 氦检仪启动
LD TR0
TIMX(550) 0906 &5  ; 氦检启动延时
; rung 18: 串口通讯异常
LD P_On
OUT TR0
AND 1559.15  ; 单元2的串口1执行标志
TIMX(550) 0907 &30  ; 氦检仪通讯异常时间
LD TR0
AND T0907  ; 氦检仪通讯异常时间
OUT 1550.03  ; 单元2串口1异常退出
@MOV(021) #0 D8100  ; 氦检仪状态(1-检漏,2-待机,3-启动,4-定标,5-错误,6-暂停)

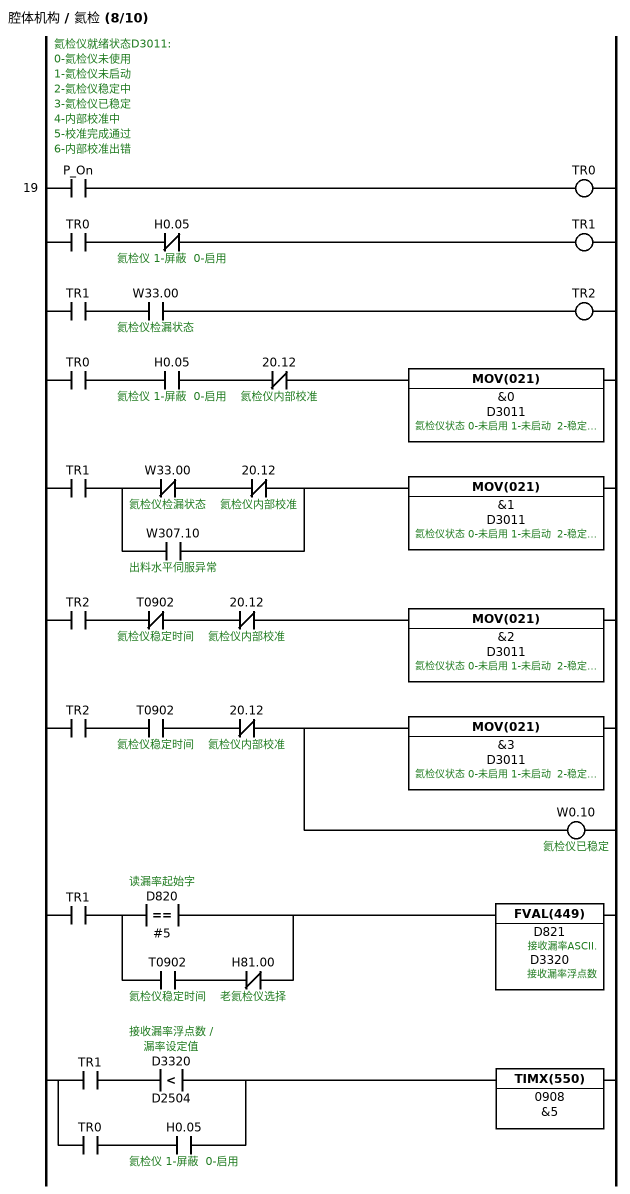
; rung 19: 氦检仪就绪状态D3011: / 0-氦检仪未使用 / 1-氦检仪未启动 / 2-氦检仪稳定中 / 3-氦检仪已稳定 / 4-内部校准中 / 5-校准完成通过 / 6-内部校准出错
LD P_On
OUT TR0
AND H0.05  ; 氦检仪 1-屏蔽  0-启用
ANDNOT 20.12  ; 氦检仪内部校准
MOV(021) &0 D3011  ; 氦检仪状态 0-未启用 1-未启动  2-稳定中 3-已稳定 4-内部校准中 5-校准完成 6-校准出错
LD TR0
ANDNOT H0.05  ; 氦检仪 1-屏蔽  0-启用
OUT TR1
LDNOT W33.00  ; 氦检仪检漏状态
ANDNOT 20.12  ; 氦检仪内部校准
OR W307.10  ; 出料水平伺服异常
ANDLD
MOV(021) &1 D3011  ; 氦检仪状态 0-未启用 1-未启动  2-稳定中 3-已稳定 4-内部校准中 5-校准完成 6-校准出错
LD TR1
AND W33.00  ; 氦检仪检漏状态
OUT TR2
ANDNOT T0902  ; 氦检仪稳定时间
ANDNOT 20.12  ; 氦检仪内部校准
MOV(021) &2 D3011  ; 氦检仪状态 0-未启用 1-未启动  2-稳定中 3-已稳定 4-内部校准中 5-校准完成 6-校准出错
LD TR2
AND T0902  ; 氦检仪稳定时间
ANDNOT 20.12  ; 氦检仪内部校准
MOV(021) &3 D3011  ; 氦检仪状态 0-未启用 1-未启动  2-稳定中 3-已稳定 4-内部校准中 5-校准完成 6-校准出错
OUT W0.10  ; 氦检仪已稳定
LD TR1
LD=(300) D820 #5  ; 读漏率起始字
LD T0902  ; 氦检仪稳定时间
ANDNOT H81.00  ; 老氦检仪选择
ORLD
ANDLD
FVAL(449) D821 D3320  ; 接收漏率ASCII., 接收漏率浮点数
LD TR1
AND<F(331) D3320 D2504  ; 接收漏率浮点数, 漏率设定值
LD TR0
AND H0.05  ; 氦检仪 1-屏蔽  0-启用
ORLD
TIMX(550) 0908 &5

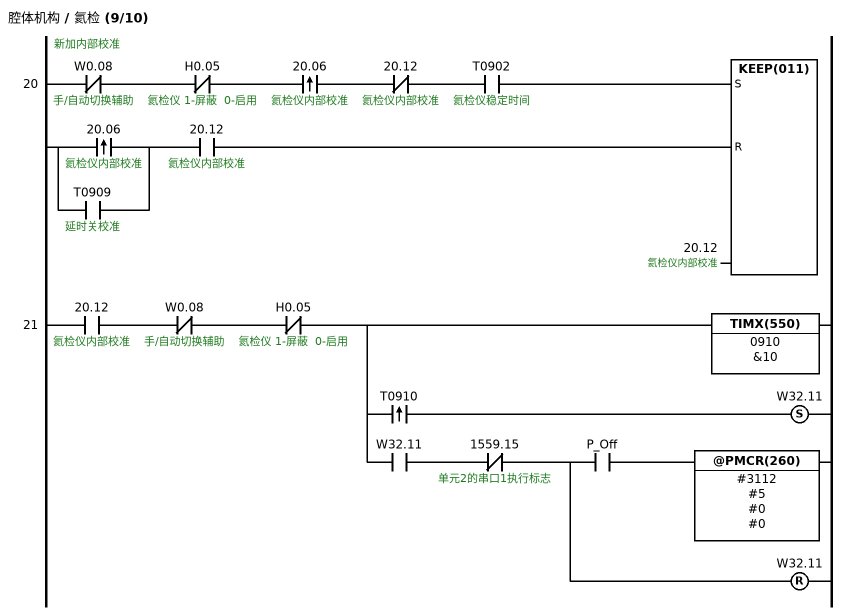
; rung 20: 新加内部校准
LDNOT W0.08  ; 手/自动切换辅助
ANDNOT H0.05  ; 氦检仪 1-屏蔽  0-启用
@AND 20.06  ; 氦检仪内部校准
ANDNOT 20.12  ; 氦检仪内部校准
AND T0902  ; 氦检仪稳定时间
@LD 20.06  ; 氦检仪内部校准
OR T0909  ; 延时关校准
AND 20.12  ; 氦检仪内部校准
KEEP(011) 20.12  ; 氦检仪内部校准
; rung 21
LD 20.12  ; 氦检仪内部校准
ANDNOT W0.08  ; 手/自动切换辅助
ANDNOT H0.05  ; 氦检仪 1-屏蔽  0-启用
OUT TR0
TIMX(550) 0910 &10
@AND T0910
SET W32.11
LD TR0
AND W32.11
ANDNOT 1559.15  ; 单元2的串口1执行标志
OUT TR0
AND P_Off
@PMCR(260) #3112 #5 #0 #0
LD TR0
RSET W32.11

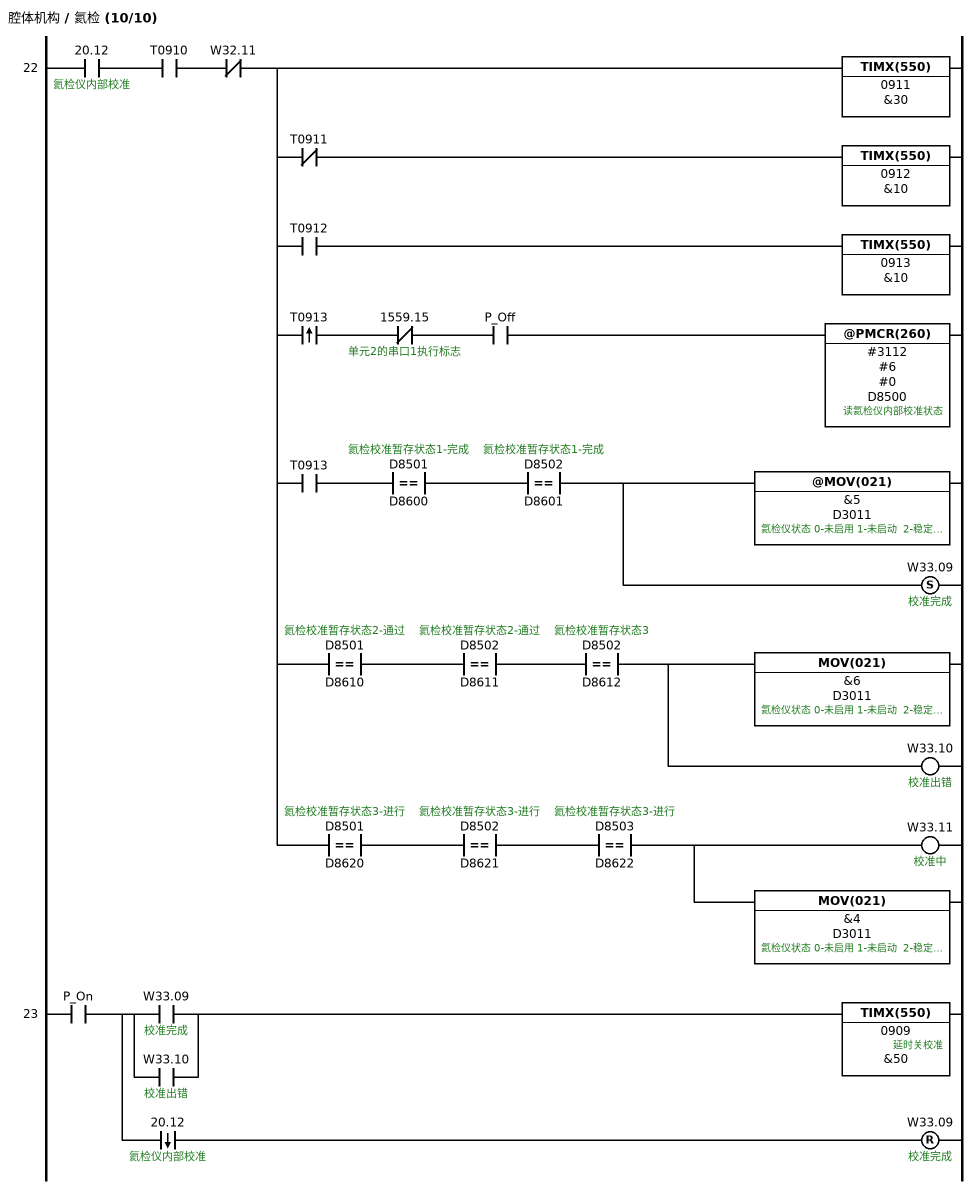
; rung 22
LD 20.12  ; 氦检仪内部校准
AND T0910
ANDNOT W32.11
OUT TR0
TIMX(550) 0911 &30
ANDNOT T0911
TIMX(550) 0912 &10
LD TR0
AND T0912
TIMX(550) 0913 &10
LD TR0
@AND T0913
ANDNOT 1559.15  ; 单元2的串口1执行标志
AND P_Off
@PMCR(260) #3112 #6 #0 D8500  ; 读氦检仪内部校准状态
LD TR0
AND T0913
AND=(300) D8501 D8600  ; 氦检校准暂存状态1-完成
AND=(300) D8502 D8601  ; 氦检校准暂存状态1-完成
@MOV(021) &5 D3011  ; 氦检仪状态 0-未启用 1-未启动  2-稳定中 3-已稳定 4-内部校准中 5-校准完成 6-校准出错
SET W33.09  ; 校准完成
LD TR0
AND=(300) D8501 D8610  ; 氦检校准暂存状态2-通过
AND=(300) D8502 D8611  ; 氦检校准暂存状态2-通过
AND=(300) D8502 D8612  ; 氦检校准暂存状态3
MOV(021) &6 D3011  ; 氦检仪状态 0-未启用 1-未启动  2-稳定中 3-已稳定 4-内部校准中 5-校准完成 6-校准出错
OUT W33.10  ; 校准出错
LD TR0
AND=(300) D8501 D8620  ; 氦检校准暂存状态3-进行
AND=(300) D8502 D8621  ; 氦检校准暂存状态3-进行
AND=(300) D8503 D8622  ; 氦检校准暂存状态3-进行
OUT W33.11  ; 校准中
MOV(021) &4 D3011  ; 氦检仪状态 0-未启用 1-未启动  2-稳定中 3-已稳定 4-内部校准中 5-校准完成 6-校准出错
; rung 23
LD P_On
OUT TR0
LD W33.09  ; 校准完成
OR W33.10  ; 校准出错
ANDLD
TIMX(550) 0909 &50  ; 延时关校准
LD TR0
%AND 20.12  ; 氦检仪内部校准
RSET W33.09  ; 校准完成

### Section _1腔体自动

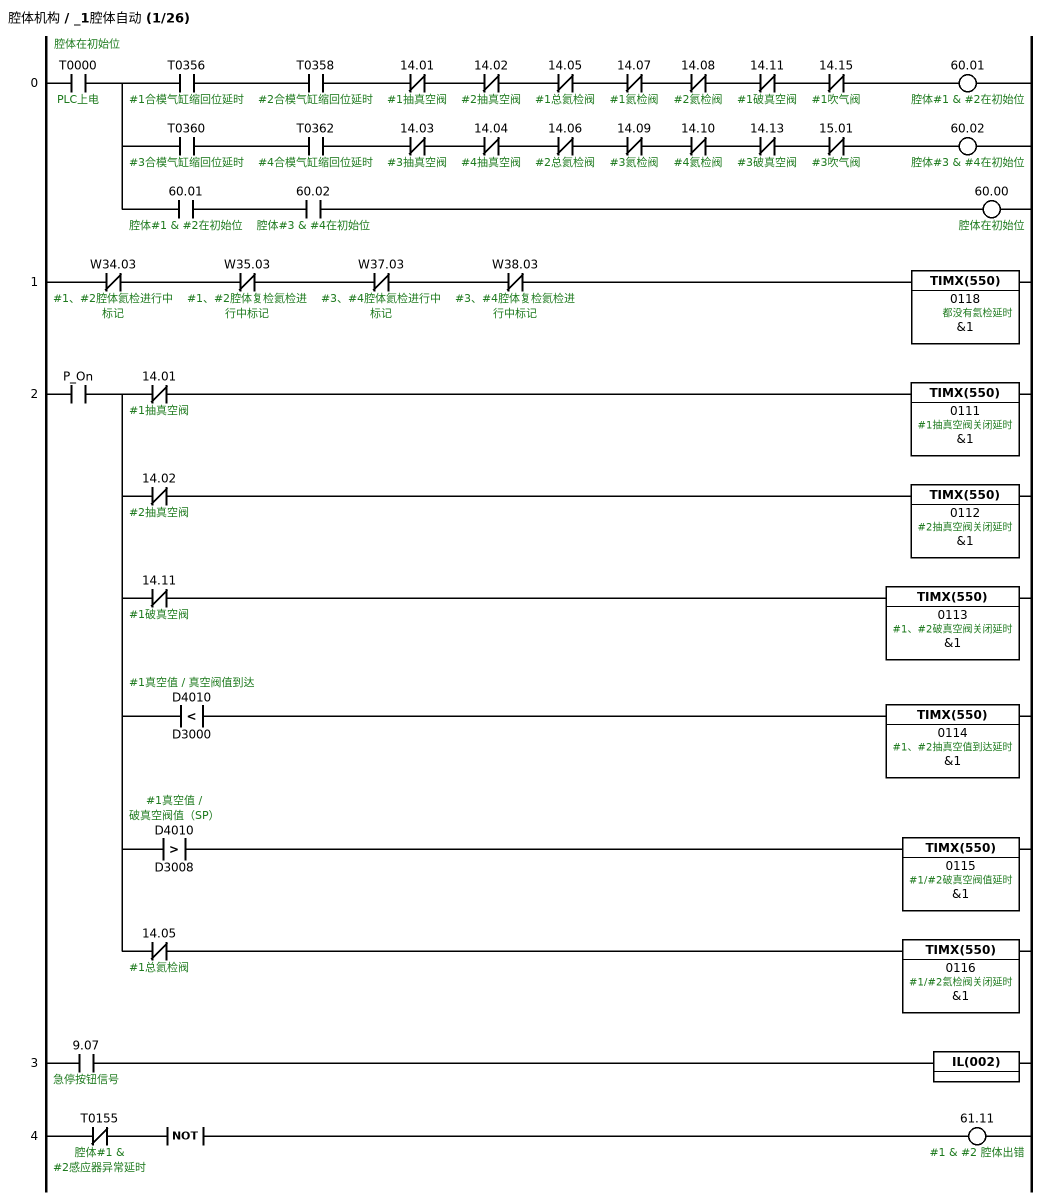
; rung 0: 腔体在初始位
LD T0000  ; PLC上电
OUT TR0
AND T0356  ; #1合模气缸缩回位延时
AND T0358  ; #2合模气缸缩回位延时
ANDNOT 14.01  ; #1抽真空阀
ANDNOT 14.02  ; #2抽真空阀
ANDNOT 14.05  ; #1总氦检阀
ANDNOT 14.07  ; #1氦检阀
ANDNOT 14.08  ; #2氦检阀
ANDNOT 14.11  ; #1破真空阀
ANDNOT 14.15  ; #1吹气阀
OUT 60.01  ; 腔体#1 & #2在初始位
LD TR0
AND T0360  ; #3合模气缸缩回位延时
AND T0362  ; #4合模气缸缩回位延时
ANDNOT 14.03  ; #3抽真空阀
ANDNOT 14.04  ; #4抽真空阀
ANDNOT 14.06  ; #2总氦检阀
ANDNOT 14.09  ; #3氦检阀
ANDNOT 14.10  ; #4氦检阀
ANDNOT 14.13  ; #3破真空阀
ANDNOT 15.01  ; #3吹气阀
OUT 60.02  ; 腔体#3 & #4在初始位
LD TR0
AND 60.01  ; 腔体#1 & #2在初始位
AND 60.02  ; 腔体#3 & #4在初始位
OUT 60.00  ; 腔体在初始位
; rung 1
LDNOT W34.03  ; #1、#2腔体氦检进行中标记
ANDNOT W35.03  ; #1、#2腔体复检氦检进行中标记
ANDNOT W37.03  ; #3、#4腔体氦检进行中标记
ANDNOT W38.03  ; #3、#4腔体复检氦检进行中标记
TIMX(550) 0118 &1  ; 都没有氦检延时
; rung 2
LD P_On
OUT TR0
ANDNOT 14.01  ; #1抽真空阀
TIMX(550) 0111 &1  ; #1抽真空阀关闭延时
LD TR0
ANDNOT 14.02  ; #2抽真空阀
TIMX(550) 0112 &1  ; #2抽真空阀关闭延时
LD TR0
ANDNOT 14.11  ; #1破真空阀
TIMX(550) 0113 &1  ; #1、#2破真空阀关闭延时
LD TR0
AND<F(331) D4010 D3000  ; #1真空值, 真空阀值到达
TIMX(550) 0114 &1  ; #1、#2抽真空值到达延时
LD TR0
AND>F(333) D4010 D3008  ; #1真空值, 破真空阀值（SP）
TIMX(550) 0115 &1  ; #1/#2破真空阀值延时
LD TR0
ANDNOT 14.05  ; #1总氦检阀
TIMX(550) 0116 &1  ; #1/#2氦检阀关闭延时
; rung 3
LD 9.07  ; 急停按钮信号
IL(002)
; rung 4
LDNOT T0155  ; 腔体#1 & #2感应器异常延时
NOT(520)
OUT 61.11  ; #1 & #2 腔体出错

